{attribute 'qualified_only'}
{attribute 'strict'}
TYPE E_RotationDirection :
(
	CW 	:= 0,
	CCW	:= 1
);
END_TYPE

(* stored: Version 1.1.0.1, ProductVersion 3.1.4024.15
   EnumerationTextList E_RotationDirection: Id {f89a10ea-c6df-4800-a3f4-949b971cf74a} *)
